// TIA Portal V15.1 export
// export: Created 2024-06-21T08:41:22.0977988Z, ExportSetting WithDefaults, DisplayName Totally Integrated Automation Portal, DisplayVersion V15.1 Update 5, DisplayName TIA Portal Openness, DisplayVersion V15.1 Update 5, DisplayName SINAMICS Startdrive Advanced, DisplayVersion V15.1, DisplayName G130, G150, S120, S150, SINAMICS MV, S210, DisplayVersion V15.1, DisplayName G110M, G120, G120C, G120D, G120P, DisplayVersion V15.1, DisplayName STEP 7 Professional, DisplayVersion V15.1 Update 5, DisplayName STEP 7 Safety, DisplayVersion V15.1, DisplayName WinCC Professional, DisplayVersion V15.1 Update 5, DisplayName SIMATIC Visualization Architect, DisplayVersion V15.1
FUNCTION "209220ZMS011Modes" : Void   // FC360, FBD
TITLE = 209220ZMS011 Modes
{ S7_Optimized_Access := 'FALSE' }
AUTHOR : VCC
FAMILY : Local
NAME : Local
VERSION : 0.1
// stored: AutoNumber false, IsIECCheckEnabled false, SetENOAutomatically False, UDAEnableTagReadback false
   VAR_OUTPUT
      O_AlarmA : Bool;   // Alarm A
      O_AlarmB : Bool;   // Alarm B
      O_AlarmC : Bool;   // Alarm C
      O_AlarmD : Bool;   // Alarm D
      O_AlarmABCondition : Bool;   // Alarms resetable
      H_IAnim : Word;   // Animation bits to Icon in WinCC
   END_VAR
   VAR_TEMP
      NotUsed : Bool;
   END_VAR
BEGIN

REGION Network 1: **** 1 - Inputs **** General Functions
   // General Functions
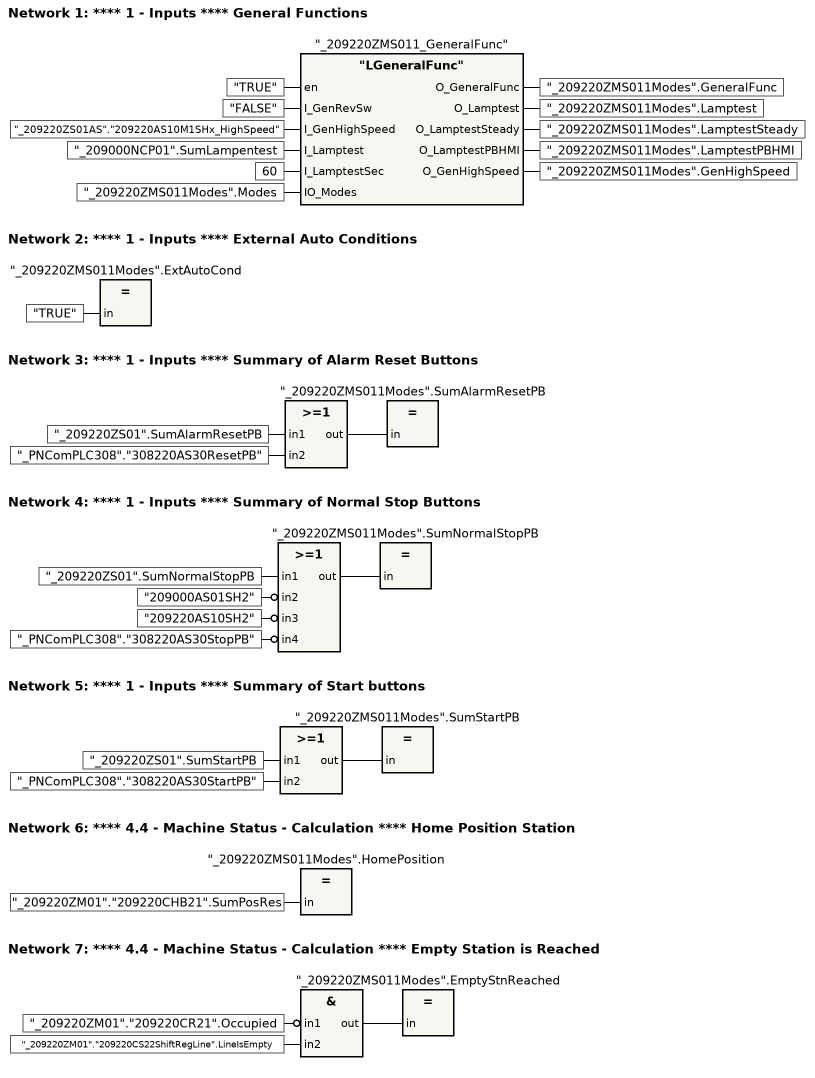
   IF "TRUE" THEN
       "_209220ZMS011_GeneralFunc"(I_GenRevSw := "FALSE",   // "LGeneralFunc"
                               I_GenHighSpeed := "_209220ZS01AS"."209220AS10M1SHx_HighSpeed",
                               I_Lamptest := "_209000NCP01".SumLampentest,
                               I_LamptestSec := 60,
                               IO_Modes := "_209220ZMS011Modes".Modes,
                               O_GeneralFunc => "_209220ZMS011Modes".GeneralFunc,
                               O_Lamptest => "_209220ZMS011Modes".Lamptest,
                               O_LamptestSteady => "_209220ZMS011Modes".LamptestSteady,
                               O_LamptestPBHMI => "_209220ZMS011Modes".LamptestPBHMI,
                               O_GenHighSpeed => "_209220ZMS011Modes".GenHighSpeed);
   END_IF;
END_REGION

REGION Network 2: **** 1 - Inputs **** External Auto Conditions
   "_209220ZMS011Modes".ExtAutoCond := "TRUE";
END_REGION

REGION Network 3: **** 1 - Inputs **** Summary of Alarm Reset Buttons
   // Summary of Alarm Reset Buttons
   "_209220ZMS011Modes".SumAlarmResetPB := "_209220ZS01".SumAlarmResetPB OR "_PNComPLC308"."308220AS30ResetPB";
END_REGION

REGION Network 4: **** 1 - Inputs **** Summary of Normal Stop Buttons
   // Summary of Normal Stop Buttons
   "_209220ZMS011Modes".SumNormalStopPB := "_209220ZS01".SumNormalStopPB OR NOT "209000AS01SH2" OR NOT "209220AS10SH2" OR NOT "_PNComPLC308"."308220AS30StopPB";
END_REGION

REGION Network 5: **** 1 - Inputs **** Summary of Start buttons
   // Summary of Start buttons
   "_209220ZMS011Modes".SumStartPB := "_209220ZS01".SumStartPB OR "_PNComPLC308"."308220AS30StartPB";
END_REGION

REGION Network 6: **** 4.4 - Machine Status - Calculation **** Home Position Station
   // Home position
   "_209220ZMS011Modes".HomePosition := "_209220ZM01"."209220CHB21".SumPosRes;
END_REGION

REGION Network 7: **** 4.4 - Machine Status - Calculation **** Empty Station is Reached
   // Empty Station
   "_209220ZMS011Modes".EmptyStnReached := NOT "_209220ZM01"."209220CR21".Occupied AND "_209220ZM01"."209220CS22ShiftRegLine".LineIsEmpty;
END_REGION

REGION Network 8: **** 4.5 - Machine Status - Modes **** Mode selector
   // Mode selector
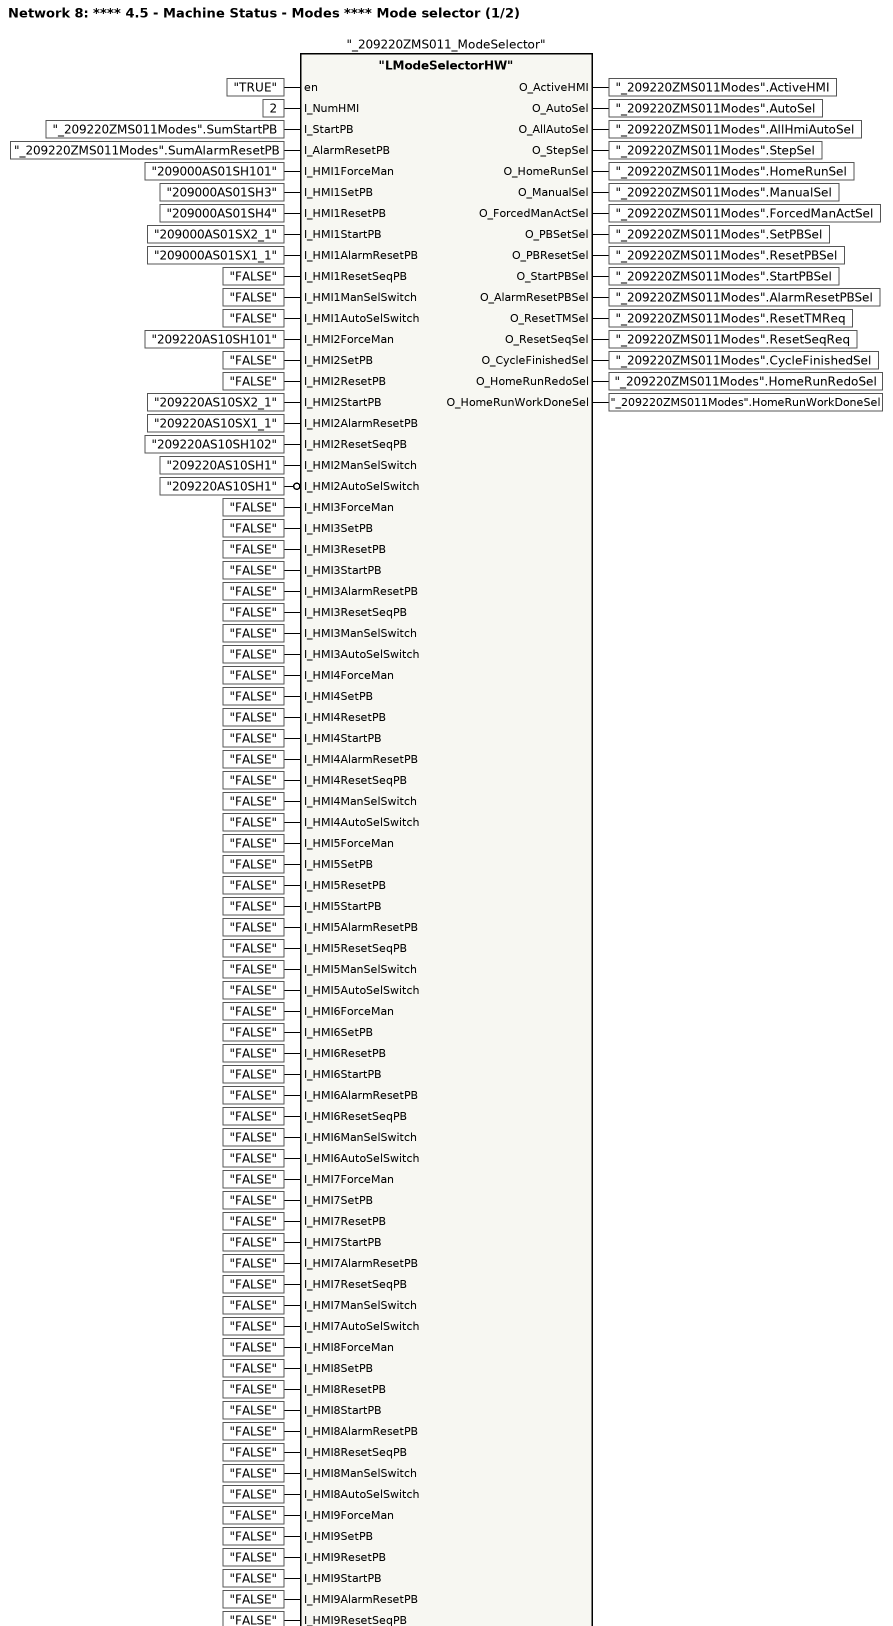
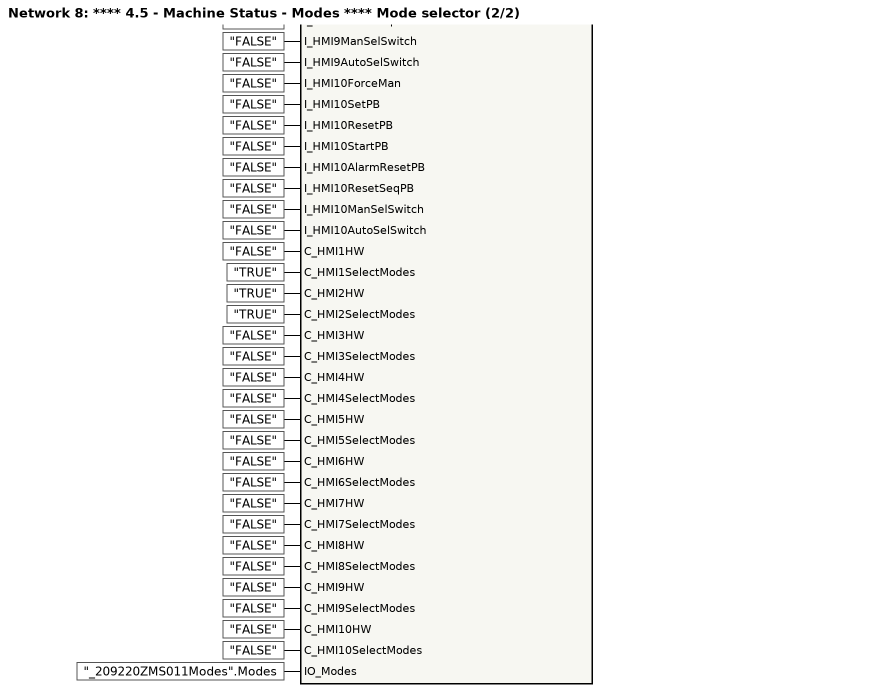
   IF "TRUE" THEN
       "_209220ZMS011_ModeSelector"(I_NumHMI := 2,   // "LModeSelectorHW"
                               I_StartPB := "_209220ZMS011Modes".SumStartPB,
                               I_AlarmResetPB := "_209220ZMS011Modes".SumAlarmResetPB,
                               I_HMI1ForceMan := "209000AS01SH101",
                               I_HMI1SetPB := "209000AS01SH3",
                               I_HMI1ResetPB := "209000AS01SH4",
                               I_HMI1StartPB := "209000AS01SX2_1",
                               I_HMI1AlarmResetPB := "209000AS01SX1_1",
                               I_HMI1ResetSeqPB := "FALSE",
                               I_HMI1ManSelSwitch := "FALSE",
                               I_HMI1AutoSelSwitch := "FALSE",
                               I_HMI2ForceMan := "209220AS10SH101",
                               I_HMI2SetPB := "FALSE",
                               I_HMI2ResetPB := "FALSE",
                               I_HMI2StartPB := "209220AS10SX2_1",
                               I_HMI2AlarmResetPB := "209220AS10SX1_1",
                               I_HMI2ResetSeqPB := "209220AS10SH102",
                               I_HMI2ManSelSwitch := "209220AS10SH1",
                               I_HMI2AutoSelSwitch := NOT "209220AS10SH1",
                               I_HMI3ForceMan := "FALSE",
                               I_HMI3SetPB := "FALSE",
                               I_HMI3ResetPB := "FALSE",
                               I_HMI3StartPB := "FALSE",
                               I_HMI3AlarmResetPB := "FALSE",
                               I_HMI3ResetSeqPB := "FALSE",
                               I_HMI3ManSelSwitch := "FALSE",
                               I_HMI3AutoSelSwitch := "FALSE",
                               I_HMI4ForceMan := "FALSE",
                               I_HMI4SetPB := "FALSE",
                               I_HMI4ResetPB := "FALSE",
                               I_HMI4StartPB := "FALSE",
                               I_HMI4AlarmResetPB := "FALSE",
                               I_HMI4ResetSeqPB := "FALSE",
                               I_HMI4ManSelSwitch := "FALSE",
                               I_HMI4AutoSelSwitch := "FALSE",
                               I_HMI5ForceMan := "FALSE",
                               I_HMI5SetPB := "FALSE",
                               I_HMI5ResetPB := "FALSE",
                               I_HMI5StartPB := "FALSE",
                               I_HMI5AlarmResetPB := "FALSE",
                               I_HMI5ResetSeqPB := "FALSE",
                               I_HMI5ManSelSwitch := "FALSE",
                               I_HMI5AutoSelSwitch := "FALSE",
                               I_HMI6ForceMan := "FALSE",
                               I_HMI6SetPB := "FALSE",
                               I_HMI6ResetPB := "FALSE",
                               I_HMI6StartPB := "FALSE",
                               I_HMI6AlarmResetPB := "FALSE",
                               I_HMI6ResetSeqPB := "FALSE",
                               I_HMI6ManSelSwitch := "FALSE",
                               I_HMI6AutoSelSwitch := "FALSE",
                               I_HMI7ForceMan := "FALSE",
                               I_HMI7SetPB := "FALSE",
                               I_HMI7ResetPB := "FALSE",
                               I_HMI7StartPB := "FALSE",
                               I_HMI7AlarmResetPB := "FALSE",
                               I_HMI7ResetSeqPB := "FALSE",
                               I_HMI7ManSelSwitch := "FALSE",
                               I_HMI7AutoSelSwitch := "FALSE",
                               I_HMI8ForceMan := "FALSE",
                               I_HMI8SetPB := "FALSE",
                               I_HMI8ResetPB := "FALSE",
                               I_HMI8StartPB := "FALSE",
                               I_HMI8AlarmResetPB := "FALSE",
                               I_HMI8ResetSeqPB := "FALSE",
                               I_HMI8ManSelSwitch := "FALSE",
                               I_HMI8AutoSelSwitch := "FALSE",
                               I_HMI9ForceMan := "FALSE",
                               I_HMI9SetPB := "FALSE",
                               I_HMI9ResetPB := "FALSE",
                               I_HMI9StartPB := "FALSE",
                               I_HMI9AlarmResetPB := "FALSE",
                               I_HMI9ResetSeqPB := "FALSE",
                               I_HMI9ManSelSwitch := "FALSE",
                               I_HMI9AutoSelSwitch := "FALSE",
                               I_HMI10ForceMan := "FALSE",
                               I_HMI10SetPB := "FALSE",
                               I_HMI10ResetPB := "FALSE",
                               I_HMI10StartPB := "FALSE",
                               I_HMI10AlarmResetPB := "FALSE",
                               I_HMI10ResetSeqPB := "FALSE",
                               I_HMI10ManSelSwitch := "FALSE",
                               I_HMI10AutoSelSwitch := "FALSE",
                               C_HMI1HW := "FALSE",
                               C_HMI1SelectModes := "TRUE",
                               C_HMI2HW := "TRUE",
                               C_HMI2SelectModes := "TRUE",
                               C_HMI3HW := "FALSE",
                               C_HMI3SelectModes := "FALSE",
                               C_HMI4HW := "FALSE",
                               C_HMI4SelectModes := "FALSE",
                               C_HMI5HW := "FALSE",
                               C_HMI5SelectModes := "FALSE",
                               C_HMI6HW := "FALSE",
                               C_HMI6SelectModes := "FALSE",
                               C_HMI7HW := "FALSE",
                               C_HMI7SelectModes := "FALSE",
                               C_HMI8HW := "FALSE",
                               C_HMI8SelectModes := "FALSE",
                               C_HMI9HW := "FALSE",
                               C_HMI9SelectModes := "FALSE",
                               C_HMI10HW := "FALSE",
                               C_HMI10SelectModes := "FALSE",
                               IO_Modes := "_209220ZMS011Modes".Modes,
                               O_ActiveHMI => "_209220ZMS011Modes".ActiveHMI,
                               O_AutoSel => "_209220ZMS011Modes".AutoSel,
                               O_AllAutoSel => "_209220ZMS011Modes".AllHmiAutoSel,
                               O_StepSel => "_209220ZMS011Modes".StepSel,
                               O_HomeRunSel => "_209220ZMS011Modes".HomeRunSel,
                               O_ManualSel => "_209220ZMS011Modes".ManualSel,
                               O_ForcedManActSel => "_209220ZMS011Modes".ForcedManActSel,
                               O_PBSetSel => "_209220ZMS011Modes".SetPBSel,
                               O_PBResetSel => "_209220ZMS011Modes".ResetPBSel,
                               O_StartPBSel => "_209220ZMS011Modes".StartPBSel,
                               O_AlarmResetPBSel => "_209220ZMS011Modes".AlarmResetPBSel,
                               O_ResetTMSel => "_209220ZMS011Modes".ResetTMReq,
                               O_ResetSeqSel => "_209220ZMS011Modes".ResetSeqReq,
                               O_CycleFinishedSel => "_209220ZMS011Modes".CycleFinishedSel,
                               O_HomeRunRedoSel => "_209220ZMS011Modes".HomeRunRedoSel,
                               O_HomeRunWorkDoneSel => "_209220ZMS011Modes".HomeRunWorkDoneSel);
   END_IF;
END_REGION

REGION Network 9: **** 4.5 - Machine Status - Modes **** Modes
   // Modes
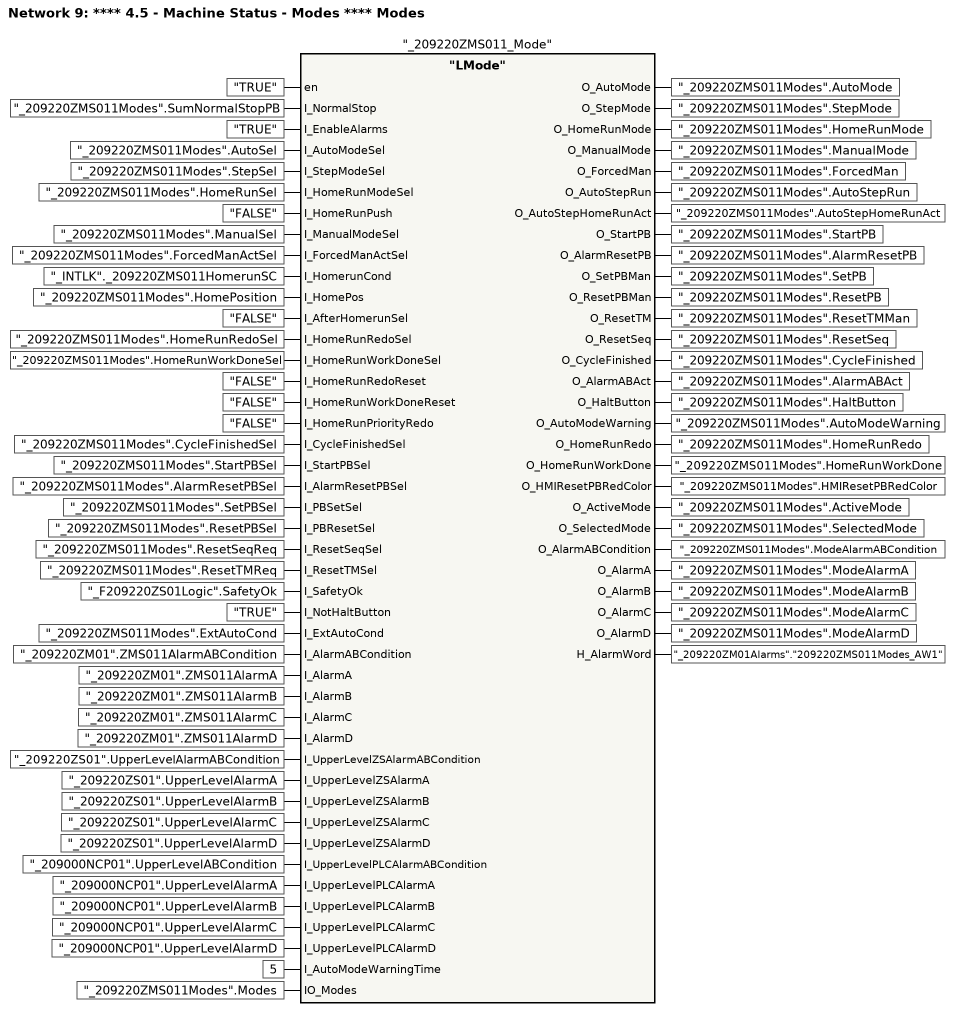
   IF "TRUE" THEN
       "_209220ZMS011_Mode"(I_NormalStop := "_209220ZMS011Modes".SumNormalStopPB,   // "LMode"
                            I_EnableAlarms := "TRUE",
                            I_AutoModeSel := "_209220ZMS011Modes".AutoSel,
                            I_StepModeSel := "_209220ZMS011Modes".StepSel,
                            I_HomeRunModeSel := "_209220ZMS011Modes".HomeRunSel,
                            I_HomeRunPush := "FALSE",
                            I_ManualModeSel := "_209220ZMS011Modes".ManualSel,
                            I_ForcedManActSel := "_209220ZMS011Modes".ForcedManActSel,
                            I_HomerunCond := "_INTLK"._209220ZMS011HomerunSC,
                            I_HomePos := "_209220ZMS011Modes".HomePosition,
                            I_AfterHomerunSel := "FALSE",
                            I_HomeRunRedoSel := "_209220ZMS011Modes".HomeRunRedoSel,
                            I_HomeRunWorkDoneSel := "_209220ZMS011Modes".HomeRunWorkDoneSel,
                            I_HomeRunRedoReset := "FALSE",
                            I_HomeRunWorkDoneReset := "FALSE",
                            I_HomeRunPriorityRedo := "FALSE",
                            I_CycleFinishedSel := "_209220ZMS011Modes".CycleFinishedSel,
                            I_StartPBSel := "_209220ZMS011Modes".StartPBSel,
                            I_AlarmResetPBSel := "_209220ZMS011Modes".AlarmResetPBSel,
                            I_PBSetSel := "_209220ZMS011Modes".SetPBSel,
                            I_PBResetSel := "_209220ZMS011Modes".ResetPBSel,
                            I_ResetSeqSel := "_209220ZMS011Modes".ResetSeqReq,
                            I_ResetTMSel := "_209220ZMS011Modes".ResetTMReq,
                            I_SafetyOk := "_F209220ZS01Logic".SafetyOk,
                            I_NotHaltButton := "TRUE",
                            I_ExtAutoCond := "_209220ZMS011Modes".ExtAutoCond,
                            I_AlarmABCondition := "_209220ZM01".ZMS011AlarmABCondition,
                            I_AlarmA := "_209220ZM01".ZMS011AlarmA,
                            I_AlarmB := "_209220ZM01".ZMS011AlarmB,
                            I_AlarmC := "_209220ZM01".ZMS011AlarmC,
                            I_AlarmD := "_209220ZM01".ZMS011AlarmD,
                            I_UpperLevelZSAlarmABCondition := "_209220ZS01".UpperLevelAlarmABCondition,
                            I_UpperLevelZSAlarmA := "_209220ZS01".UpperLevelAlarmA,
                            I_UpperLevelZSAlarmB := "_209220ZS01".UpperLevelAlarmB,
                            I_UpperLevelZSAlarmC := "_209220ZS01".UpperLevelAlarmC,
                            I_UpperLevelZSAlarmD := "_209220ZS01".UpperLevelAlarmD,
                            I_UpperLevelPLCAlarmABCondition := "_209000NCP01".UpperLevelABCondition,
                            I_UpperLevelPLCAlarmA := "_209000NCP01".UpperLevelAlarmA,
                            I_UpperLevelPLCAlarmB := "_209000NCP01".UpperLevelAlarmB,
                            I_UpperLevelPLCAlarmC := "_209000NCP01".UpperLevelAlarmC,
                            I_UpperLevelPLCAlarmD := "_209000NCP01".UpperLevelAlarmD,
                            I_AutoModeWarningTime := 5,
                            IO_Modes := "_209220ZMS011Modes".Modes,
                            O_AutoMode => "_209220ZMS011Modes".AutoMode,
                            O_StepMode => "_209220ZMS011Modes".StepMode,
                            O_HomeRunMode => "_209220ZMS011Modes".HomeRunMode,
                            O_ManualMode => "_209220ZMS011Modes".ManualMode,
                            O_ForcedMan => "_209220ZMS011Modes".ForcedMan,
                            O_AutoStepRun => "_209220ZMS011Modes".AutoStepRun,
                            O_AutoStepHomeRunAct => "_209220ZMS011Modes".AutoStepHomeRunAct,
                            O_StartPB => "_209220ZMS011Modes".StartPB,
                            O_AlarmResetPB => "_209220ZMS011Modes".AlarmResetPB,
                            O_SetPBMan => "_209220ZMS011Modes".SetPB,
                            O_ResetPBMan => "_209220ZMS011Modes".ResetPB,
                            O_ResetTM => "_209220ZMS011Modes".ResetTMMan,
                            O_ResetSeq => "_209220ZMS011Modes".ResetSeq,
                            O_CycleFinished => "_209220ZMS011Modes".CycleFinished,
                            O_AlarmABAct => "_209220ZMS011Modes".AlarmABAct,
                            O_HaltButton => "_209220ZMS011Modes".HaltButton,
                            O_AutoModeWarning => "_209220ZMS011Modes".AutoModeWarning,
                            O_HomeRunRedo => "_209220ZMS011Modes".HomeRunRedo,
                            O_HomeRunWorkDone => "_209220ZMS011Modes".HomeRunWorkDone,
                            O_HMIResetPBRedColor => "_209220ZMS011Modes".HMIResetPBRedColor,
                            O_ActiveMode => "_209220ZMS011Modes".ActiveMode,
                            O_SelectedMode => "_209220ZMS011Modes".SelectedMode,
                            O_AlarmABCondition => "_209220ZMS011Modes".ModeAlarmABCondition,
                            O_AlarmA => "_209220ZMS011Modes".ModeAlarmA,
                            O_AlarmB => "_209220ZMS011Modes".ModeAlarmB,
                            O_AlarmC => "_209220ZMS011Modes".ModeAlarmC,
                            O_AlarmD => "_209220ZMS011Modes".ModeAlarmD,
                            H_AlarmWord => "_209220ZM01Alarms"."209220ZMS011Modes_AW1");
   END_IF;
END_REGION

REGION Network 10: **** 4.5 - Machine Status - Modes **** Production Modes
   // Production Modes
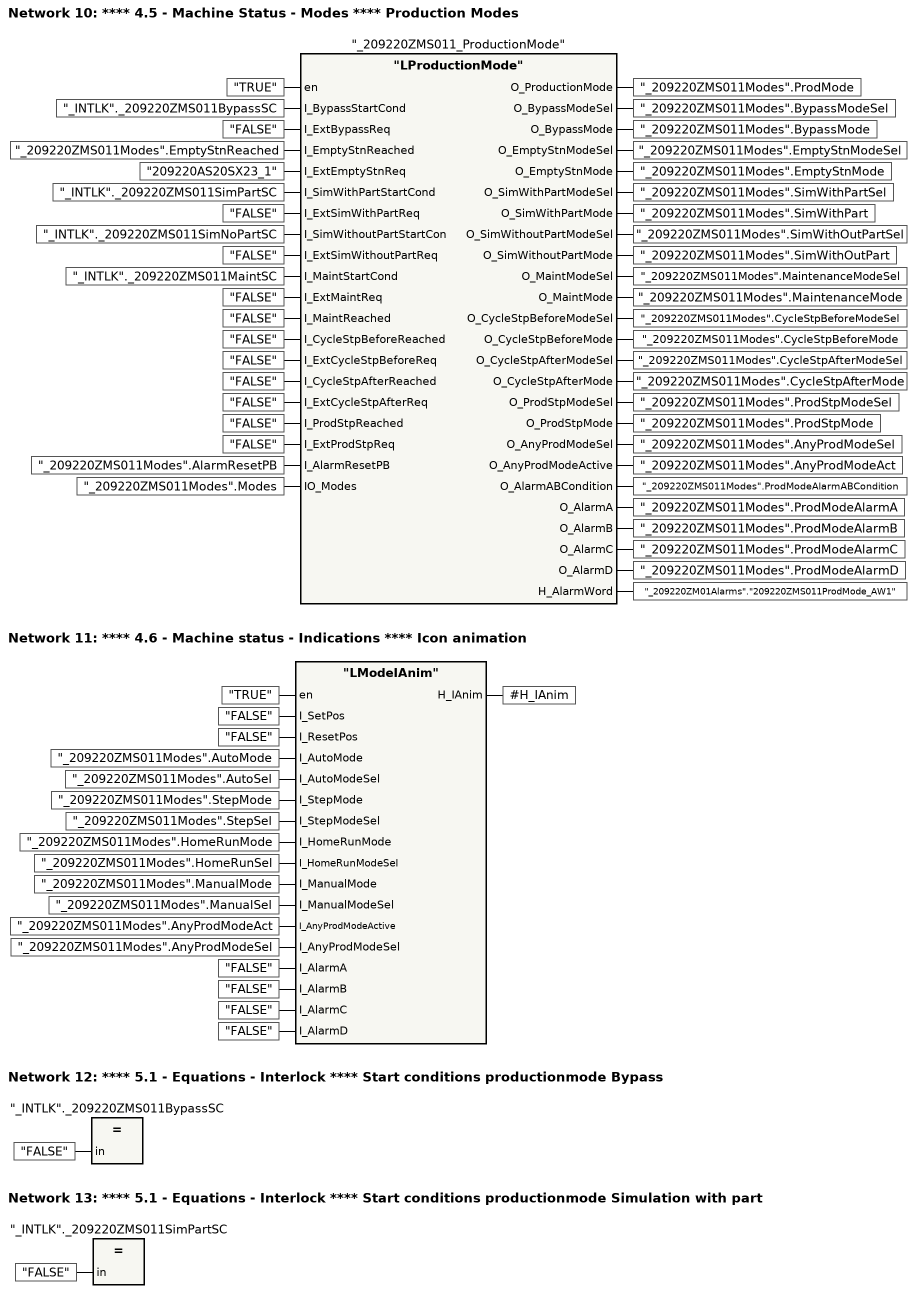
   IF "TRUE" THEN
       "_209220ZMS011_ProductionMode"(I_BypassStartCond := "_INTLK"._209220ZMS011BypassSC,   // "LProductionMode"
                               I_ExtBypassReq := "FALSE",
                               I_EmptyStnReached := "_209220ZMS011Modes".EmptyStnReached,
                               I_ExtEmptyStnReq := "209220AS20SX23_1",
                               I_SimWithPartStartCond := "_INTLK"._209220ZMS011SimPartSC,
                               I_ExtSimWithPartReq := "FALSE",
                               I_SimWithoutPartStartCon := "_INTLK"._209220ZMS011SimNoPartSC,
                               I_ExtSimWithoutPartReq := "FALSE",
                               I_MaintStartCond := "_INTLK"._209220ZMS011MaintSC,
                               I_ExtMaintReq := "FALSE",
                               I_MaintReached := "FALSE",
                               I_CycleStpBeforeReached := "FALSE",
                               I_ExtCycleStpBeforeReq := "FALSE",
                               I_CycleStpAfterReached := "FALSE",
                               I_ExtCycleStpAfterReq := "FALSE",
                               I_ProdStpReached := "FALSE",
                               I_ExtProdStpReq := "FALSE",
                               I_AlarmResetPB := "_209220ZMS011Modes".AlarmResetPB,
                               IO_Modes := "_209220ZMS011Modes".Modes,
                               O_ProductionMode => "_209220ZMS011Modes".ProdMode,
                               O_BypassModeSel => "_209220ZMS011Modes".BypassModeSel,
                               O_BypassMode => "_209220ZMS011Modes".BypassMode,
                               O_EmptyStnModeSel => "_209220ZMS011Modes".EmptyStnModeSel,
                               O_EmptyStnMode => "_209220ZMS011Modes".EmptyStnMode,
                               O_SimWithPartModeSel => "_209220ZMS011Modes".SimWithPartSel,
                               O_SimWithPartMode => "_209220ZMS011Modes".SimWithPart,
                               O_SimWithoutPartModeSel => "_209220ZMS011Modes".SimWithOutPartSel,
                               O_SimWithoutPartMode => "_209220ZMS011Modes".SimWithOutPart,
                               O_MaintModeSel => "_209220ZMS011Modes".MaintenanceModeSel,
                               O_MaintMode => "_209220ZMS011Modes".MaintenanceMode,
                               O_CycleStpBeforeModeSel => "_209220ZMS011Modes".CycleStpBeforeModeSel,
                               O_CycleStpBeforeMode => "_209220ZMS011Modes".CycleStpBeforeMode,
                               O_CycleStpAfterModeSel => "_209220ZMS011Modes".CycleStpAfterModeSel,
                               O_CycleStpAfterMode => "_209220ZMS011Modes".CycleStpAfterMode,
                               O_ProdStpModeSel => "_209220ZMS011Modes".ProdStpModeSel,
                               O_ProdStpMode => "_209220ZMS011Modes".ProdStpMode,
                               O_AnyProdModeSel => "_209220ZMS011Modes".AnyProdModeSel,
                               O_AnyProdModeActive => "_209220ZMS011Modes".AnyProdModeAct,
                               O_AlarmABCondition => "_209220ZMS011Modes".ProdModeAlarmABCondition,
                               O_AlarmA => "_209220ZMS011Modes".ProdModeAlarmA,
                               O_AlarmB => "_209220ZMS011Modes".ProdModeAlarmB,
                               O_AlarmC => "_209220ZMS011Modes".ProdModeAlarmC,
                               O_AlarmD => "_209220ZMS011Modes".ProdModeAlarmD,
                               H_AlarmWord => "_209220ZM01Alarms"."209220ZMS011ProdMode_AW1");
   END_IF;
END_REGION

REGION Network 11: **** 4.6 - Machine status - Indications **** Icon animation
   // Icon animation
   IF "TRUE" THEN
       "LModeIAnim"(I_SetPos := "FALSE",
                    I_ResetPos := "FALSE",
                    I_AutoMode := "_209220ZMS011Modes".AutoMode,
                    I_AutoModeSel := "_209220ZMS011Modes".AutoSel,
                    I_StepMode := "_209220ZMS011Modes".StepMode,
                    I_StepModeSel := "_209220ZMS011Modes".StepSel,
                    I_HomeRunMode := "_209220ZMS011Modes".HomeRunMode,
                    I_HomeRunModeSel := "_209220ZMS011Modes".HomeRunSel,
                    I_ManualMode := "_209220ZMS011Modes".ManualMode,
                    I_ManualModeSel := "_209220ZMS011Modes".ManualSel,
                    I_AnyProdModeActive := "_209220ZMS011Modes".AnyProdModeAct,
                    I_AnyProdModeSel := "_209220ZMS011Modes".AnyProdModeSel,
                    I_AlarmA := "FALSE",
                    I_AlarmB := "FALSE",
                    I_AlarmC := "FALSE",
                    I_AlarmD := "FALSE",
                    H_IAnim => #H_IAnim);
   END_IF;
END_REGION

REGION Network 12: **** 5.1 - Equations - Interlock **** Start conditions productionmode Bypass
   // Start conditions productionmode
   // Bypass
   "_INTLK"._209220ZMS011BypassSC := "FALSE";
END_REGION

REGION Network 13: **** 5.1 - Equations - Interlock **** Start conditions productionmode Simulation with part
   // Start conditions productionmode
   // Simulation with part
   "_INTLK"._209220ZMS011SimPartSC := "FALSE";
END_REGION

REGION Network 14: **** 5.1 - Equations - Interlock **** Start conditions productionmode Simulation without part
   // Start conditions productionmode
   // Simulation without part
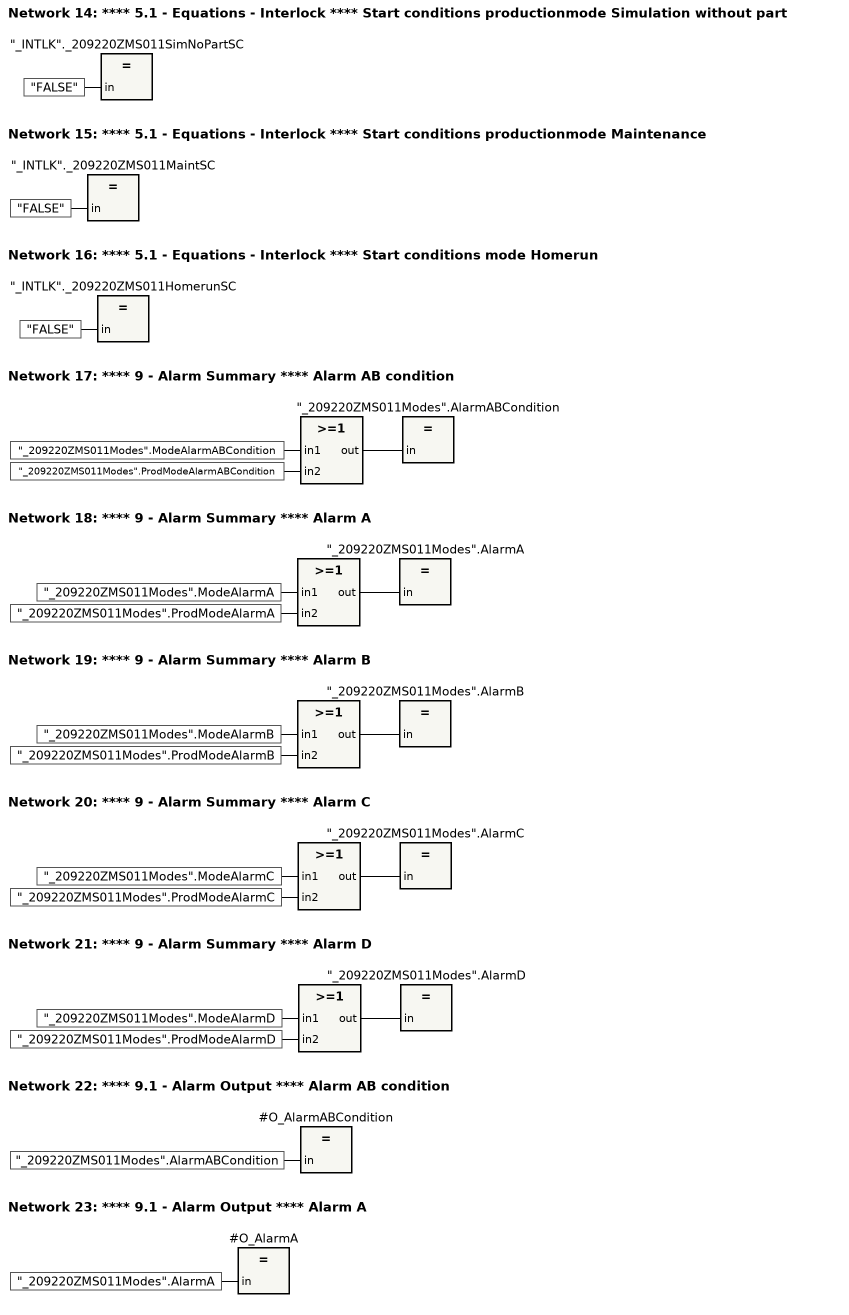
   "_INTLK"._209220ZMS011SimNoPartSC := "FALSE";
END_REGION

REGION Network 15: **** 5.1 - Equations - Interlock **** Start conditions productionmode Maintenance
   // Start conditions productionmode
   // Maintenance
   "_INTLK"._209220ZMS011MaintSC := "FALSE";
END_REGION

REGION Network 16: **** 5.1 - Equations - Interlock **** Start conditions mode Homerun
   // Start conditions mode
   // Homerun
   "_INTLK"._209220ZMS011HomerunSC := "FALSE";
END_REGION

REGION Network 17: **** 9 - Alarm Summary **** Alarm AB condition
   // Alarm AB condition
   "_209220ZMS011Modes".AlarmABCondition := "_209220ZMS011Modes".ModeAlarmABCondition OR "_209220ZMS011Modes".ProdModeAlarmABCondition;
END_REGION

REGION Network 18: **** 9 - Alarm Summary **** Alarm A
   // Summary of alarms A
   "_209220ZMS011Modes".AlarmA := "_209220ZMS011Modes".ModeAlarmA OR "_209220ZMS011Modes".ProdModeAlarmA;
END_REGION

REGION Network 19: **** 9 - Alarm Summary **** Alarm B
   // Summary of alarms B
   "_209220ZMS011Modes".AlarmB := "_209220ZMS011Modes".ModeAlarmB OR "_209220ZMS011Modes".ProdModeAlarmB;
END_REGION

REGION Network 20: **** 9 - Alarm Summary **** Alarm C
   // Summary of alarms C
   "_209220ZMS011Modes".AlarmC := "_209220ZMS011Modes".ModeAlarmC OR "_209220ZMS011Modes".ProdModeAlarmC;
END_REGION

REGION Network 21: **** 9 - Alarm Summary **** Alarm D
   // Summary of alarms D
   "_209220ZMS011Modes".AlarmD := "_209220ZMS011Modes".ModeAlarmD OR "_209220ZMS011Modes".ProdModeAlarmD;
END_REGION

REGION Network 22: **** 9.1 - Alarm Output **** Alarm AB condition
   // Alarm AB condition
   #O_AlarmABCondition := "_209220ZMS011Modes".AlarmABCondition;
END_REGION

REGION Network 23: **** 9.1 - Alarm Output **** Alarm A
   // Summary of alarms A
   #O_AlarmA := "_209220ZMS011Modes".AlarmA;
END_REGION

REGION Network 24: **** 9.1 - Alarm Output **** Alarm B
   // Summary of alarms B
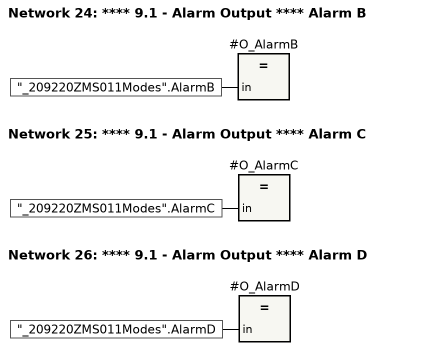
   #O_AlarmB := "_209220ZMS011Modes".AlarmB;
END_REGION

REGION Network 25: **** 9.1 - Alarm Output **** Alarm C
   // Summary of alarms C
   #O_AlarmC := "_209220ZMS011Modes".AlarmC;
END_REGION

REGION Network 26: **** 9.1 - Alarm Output **** Alarm D
   // Summary of alarms D
   #O_AlarmD := "_209220ZMS011Modes".AlarmD;
END_REGION
END_FUNCTION
